Fanuc KAREL source: kb00192.KL

-- PROVISIONAL review KL for V1013-1; original PC SHA256 6bb8237e6c9ee9c53d4e3899567e548ecf7a9bca6632220358625d738b8daaac
-- Incomplete behavior may be omitted. Consult companion uncertainty JSON. Do not deploy.
PROGRAM KB00192
%NOLOCKGROUP
VAR
  P1 : REAL
  RESULT : INTEGER
BEGIN
  -- UNRESOLVED_PC offsets 5-16; opcodes 2E,23
  -- UNRESOLVED_PC offsets 21-36; opcodes 27,22,76,23
  -- UNRESOLVED_PC offsets 41-45; opcodes 7F
END KB00192
